// TwinCAT 3 PLC project StageUtils
// Title: StageUtils
// Company: _
// Author: Krystian Lis et al.
// ProjectVersion: 4.0.0
// Description: Various Stage related utilities
// ProgramVersion: 3.1.4026.18
// libraries:
//   Tc2_Standard, * (Beckhoff Automation GmbH)
//   Tc2_System, * (Beckhoff Automation GmbH)
// project tree:
//   Color/ Argb.TcDUT, BuildArgb.TcPOU, Argbb.TcPOU
//   Color/Itf/ I_Argbb.TcIO
//   Math/ Math.TcPOU
//   Time/ GetTaskCycleTime.TcPOU, GetUnixTime.TcPOU
// real-time tasks:
//   TASK Example: cycle T#10ms, priority 20, ADS port 350
//   TASK Test: cycle T#10ms, priority 21, ADS port 351
//   TASK VISU_TASK: cycle T#200000us, priority 30, ADS port 352

// ---- Color/Argb.TcDUT
(*
A DWORD alias type to be used with PLC HMI. Encodes ARGB value.
*)
TYPE Argb : DWORD; END_TYPE

// ---- Color/Itf/I_Argbb.TcIO
(*
Provides methods and properties to operate on RGBA value.
*)
INTERFACE I_Argbb

(*
ALPHA channel
*)
PROPERTY Alpha : BYTE
GET
END_GET
SET
END_SET
END_PROPERTY

(*
BLUE component
*)
PROPERTY Blue : BYTE
GET
END_GET
SET
END_SET
END_PROPERTY

(*
Clones other components of I_RgbaColor interface.
*)
METHOD Clone
VAR_INPUT
	iColor	: I_Argbb;
END_VAR
END_METHOD

(*
GREEN component
*)
PROPERTY Green : BYTE
GET
END_GET
SET
END_SET
END_PROPERTY

(*
Compute single Color value from RGBA components when used as getter.
Sets RGBA values by extracting components from a single Color value.
*)
PROPERTY Raw : Argb
GET
END_GET
SET
END_SET
END_PROPERTY

(*
RED component
*)
PROPERTY Red : BYTE
GET
END_GET
SET
END_SET
END_PROPERTY

(*
Set each RGBA component value separately.
*)
METHOD Set
VAR_INPUT
	nRed: USINT;
	nGreen: USINT;
	nBlue: USINT;
	nAlpha: USINT;
END_VAR
END_METHOD

END_INTERFACE

// ---- Color/BuildArgb.TcPOU
(*
	Returns raw RGBA value from components.
*)
FUNCTION BuildArgb : Argb
VAR_INPUT
	nRed: USINT;
	nGreen: USINT;
	nBlue: USINT;
	nAlpha: USINT;
END_VAR

BuildArgb := USINT_TO_UDINT(nBlue) OR
			SHL(USINT_TO_UDINT(nGreen), 8) OR
			SHL(USINT_TO_UDINT(nRed), 16) OR
			SHL(USINT_TO_UDINT(nAlpha), 24);

END_FUNCTION

// ---- Color/Argbb.TcPOU
(*
Provides methods and properties to operate on RGBA value.
*)
FUNCTION_BLOCK Argbb IMPLEMENTS I_Argbb
VAR
	_r: BYTE;
	_g: BYTE;
	_b: BYTE;
	_a: BYTE;
END_VAR

(*
ALPHA channel
*)
PROPERTY Alpha : BYTE
GET
Alpha := _a;
END_GET
SET
_a := Alpha;
END_SET
END_PROPERTY

(*
BLUE component
*)
PROPERTY Blue : BYTE
GET
Blue := _b;
END_GET
SET
_b := Blue;
END_SET
END_PROPERTY

(*
Clones other components of I_RgbaColor interface.
*)
METHOD Clone
VAR_INPUT
	iColor	: I_Argbb;
END_VAR
IF iColor = 0 THEN
	RETURN;
END_IF

_r := iColor.Red;
_b := iColor.Blue;
_g := iColor.Green;
_a := iColor.Alpha;
END_METHOD

{attribute 'hide'}
METHOD FB_init : BOOL
VAR_INPUT
	bInitRetains : BOOL;
	bInCopyCode : BOOL;
	nRed: USINT;
	nGreen: USINT;
	nBlue: USINT;
	nAlpha: USINT;
END_VAR
Set(nRed, nGreen, nBlue, nAlpha);
END_METHOD

(*
GREEN component
*)
PROPERTY Green : BYTE
GET
Green := _g;
END_GET
SET
_g := Green;
END_SET
END_PROPERTY

(*
Compute single Color value from RGBA components when used as getter.
Sets RGBA values by extracting components from a single Color value.
*)
PROPERTY Raw : Argb
GET
Raw := 	USINT_TO_UDINT(_b) OR
			SHL(USINT_TO_UDINT(_g), 8) OR
			SHL(USINT_TO_UDINT(_r), 16) OR
			SHL(USINT_TO_UDINT(_a), 24);
END_GET
SET
_b := UDINT_TO_USINT(Raw AND 16#FF);
_g := UDINT_TO_USINT(SHR(Raw, 8) AND 16#FF);
_r := UDINT_TO_USINT(SHR(Raw, 16) AND 16#FF);
_a := UDINT_TO_USINT(SHR(Raw, 24) AND 16#FF);
END_SET
END_PROPERTY

(*
RED component
*)
PROPERTY Red : BYTE
GET
Red := _r;
END_GET
SET
_r := Red;
END_SET
END_PROPERTY

(*
Set each RGBA component value separately.
*)
METHOD Set
VAR_INPUT
	nRed: USINT;
	nGreen: USINT;
	nBlue: USINT;
	nAlpha: USINT;
END_VAR
_r := nRed;
_g := nGreen;
_b := nBlue;
_a := nAlpha;
END_METHOD

END_FUNCTION_BLOCK

// ---- Math/Math.TcPOU
(*Provides various mathematical functions*)
PROGRAM Math
VAR
END_VAR

(* 
    Time-compensated smoothing coefficient. 
    Alpha = 1 - (1 - B)^dt
*)
METHOD ExptDecay : LREAL
VAR_INPUT
    rBlendFactor : LREAL;   // In [0, 1] — how fast to blend toward input
    rDeltaTime   : LREAL := 0.01;   // In seconds
END_VAR
rBlendFactor := LIMIT(0.0, rBlendFactor, 1.0);
rDeltaTime   := MAX(rDeltaTime, 0.0);
ExptDecay := LIMIT(0.0, 1.0 - EXPT(1.0 - rBlendFactor, rDeltaTime), 1.0);
END_METHOD

(*
Allows for value scalling.
Returns 0 when rMaxX - rMinX = 0.
*)
METHOD LinearScale : LREAL
VAR_INPUT
	rX				: LREAL;
	rMinX			: LREAL;
	rMaxX			: LREAL;
	rMinY			: LREAL := 0;
	rMaxY			: LREAL := 1;
END_VAR
VAR
	_rDnmtr			: LREAL := rMaxX - rMinX;
END_VAR
IF _rDnmtr <> 0 THEN
	LinearScale := rMinY + ((rX - rMinX)/_rDnmtr) * (rMaxY - rMinY);
END_IF
END_METHOD

(*
First-order low pass filter.
Yt = Xt * Coeff + Y(t-1) * (1- Coeff)
*)
METHOD LowPassFilter : LREAL
VAR_INPUT
	rX				: LREAL;
	rPrvY			: LREAL;
	
	rCoefficient	: LREAL;
END_VAR
LowPassFilter := rX * rCoefficient + rPrvY * (1 - rCoefficient);
END_METHOD

(*
Generates random number every time is called.
*)
METHOD Random : LREAL
VAR_STAT
	_nSeed		: INT;
END_VAR
VAR
	_drand		: Tc2_System.DRAND;
END_VAR
_drand(Seed := _nSeed, Num => Random);
_nSeed := _nSeed + 1;
END_METHOD

END_PROGRAM

// ---- Time/GetTaskCycleTime.TcPOU
(*
	Get task cycle time in seconds.
*)
FUNCTION GetTaskCycleTime : LREAL
VAR_IN_OUT CONSTANT
	taskInfo: ARRAY[*] OF PlcTaskSystemInfo; // Just assign _TaskInfo as _TaskInfo cannot be accessed from lib :(
END_VAR

GetTaskCycleTime := UDINT_TO_LREAL(taskInfo[TC2_System.GETCURTASKINDEXEX()].CycleTime) / 10_000_000;

END_FUNCTION

// ---- Time/GetUnixTime.TcPOU
(*
Generates TIME in 100ns since 1ST January 1970.
Bases on Tc2_System.F_GetSystemTime FUNCTION.
The result can be adjusted through the nOffset variable.
*)
FUNCTION GetUnixTime : ULINT
VAR_INPUT
	nOffset : LINT := 0;
END_VAR
VAR
END_VAR

GetUnixTime := Tc2_System.F_GetSystemTime() - LINT_TO_ULINT(11_644_473_678_000_000_0 + nOffset);

END_FUNCTION
